FUNCTION_BLOCK TEST_LOGS (* Test logarithmic functions *)
  (* Standard: 61499-1 *)
  (* Version 0.0, 2006-09-05, JHC, Holobloc Inc *)
  (* Compiler header: package fb.rt.test; *)
  (* Compiler classdef: SimpleFB *)
  (* Compiler Java Sun JDK 1.5.0 *)
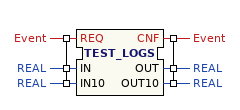
  EVENT_INPUT
    REQ WITH IN, IN10; (* Normal Execution Request *)
  END_EVENT
  EVENT_OUTPUT
    CNF WITH OUT, OUT10; (* Execution Confirmation *)
  END_EVENT
  VAR_INPUT
    IN : REAL; (* Input value for log, exp *)
    IN10 : REAL; (* Input for base 10 log *)
  END_VAR
  VAR_OUTPUT
    OUT : REAL; (* exp(ln(IN)) *)
    OUT10 : REAL; (* 10**(log10(IN10)) *)
  END_VAR
  ALGORITHM REQ IN FBD: (* Normally executed algorithm *)
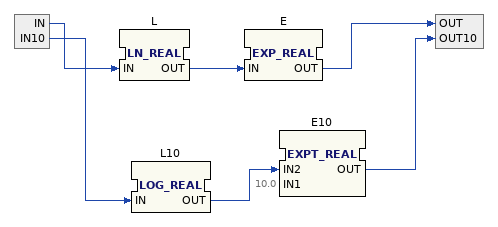
    FBS
      L : LN_REAL;
      E : EXP_REAL;
      L10 : LOG_REAL;
      E10 : EXPT_REAL(IN1 := 10.0);
    END_FBS
    DATA_CONNECTIONS
      IN TO L.IN;
      L.OUT TO E.IN;
      E.OUT TO OUT;
      IN10 TO L10.IN;
      L10.OUT TO E10.IN2;
      E10.OUT TO OUT10;
    END_CONNECTIONS
  END_ALGORITHM
END_FUNCTION_BLOCK
